FUNCTION_BLOCK FB_CintaTraer
VAR_INPUT
	TiempoEntradaPale: TIME := T#2S;
END_VAR
VAR_OUTPUT
END_VAR
VAR
	PM AT %I*: BOOL; (*pulsador de marcha*)
	pp AT %I*: BOOL; (* presencia de pale *)
	
	LM AT %Q*: BOOL; (*Lampara de marcha*)
	RUN AT %Q*: BOOL; (*activa motor*)
	
END_VAR

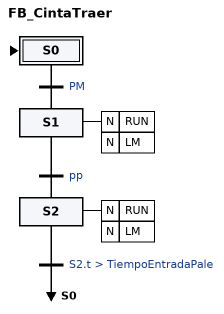
INITIAL_STEP S0:
END_STEP
TRANSITION FROM S0 TO S1
    := PM;
END_TRANSITION
STEP S1:
    RUN(N);
    LM(N);
END_STEP
TRANSITION FROM S1 TO S2
    := pp;
END_TRANSITION
STEP S2:
    RUN(N);
    LM(N);
END_STEP
TRANSITION FROM S2 TO S0
    := S2.t > TiempoEntradaPale;
END_TRANSITION

END_FUNCTION_BLOCK

(* stored: Version 1.1.0.1, ProductVersion 3.1.4024.12
   POU FB_CintaTraer: Id {7593a2a1-0097-4654-8801-4c746e83e6cf}, SpecialFunc None *)
